TYPE ST_Record :
STRUCT
    nID        : LINT;
    sName      : STRING;
    nSensor1   : REAL;
    nSensor2   : REAL;
END_STRUCT
END_TYPE

(* stored: Version 1.1.0.1, ProductVersion 3.1.4022.12
   DUT ST_Record: Id {08d1b38a-93f8-45df-89fb-bc356996c62d} *)
